// TIA Portal V20 export
// export: Created 2026-04-11T06:02:30.3000728Z, ExportSetting WithDefaults, DisplayName Totally Integrated Automation Portal, DisplayVersion V20, DisplayName TIA Portal Openness, DisplayVersion V20, DisplayName TIA Portal Version Control Interface, DisplayVersion V20, DisplayName STEP 7 Professional, DisplayVersion V20, DisplayName STEP 7 Safety, DisplayVersion V20, DisplayName WinCC Basic/Comfort/Advanced, DisplayVersion V20, DisplayName WinCC Unified, DisplayVersion V20
TYPE "udtHMI_AnalogValveControl"
// stored: IsFailsafeCompliant false
   STRUCT
      iMode : Int;   // Current mode
      iErrorCode { ExternalWritable := 'False'} : Int;   // Error code
      iStatus { ExternalWritable := 'False'} : Int;   // Color status for HMI
      rManualSP { S7_SetPoint := 'True'} : Real;   // Set point for manual mode
      rAutoSP { ExternalWritable := 'False'} : Real;   // Set point for automatic mode
      rEstopSP { S7_SetPoint := 'True'} : Real;   // Set point for an e-stop condition, if selected
      rActual { ExternalWritable := 'False'} : Real;   // Actual value
      bPB_ResetError : Bool;   // PB Reset errors
      bPBEN_ResetError { ExternalWritable := 'False'} : Bool;   // PB reset errors enable
      bError { ExternalWritable := 'False'} : Bool;   // Overall error
      bInterlock { ExternalWritable := 'False'} : Bool;   // Valve Interlocked
      iEstopFunction { S7_SetPoint := 'True'} : Int;   // Enum of E-Stop repsonse (Estop.xxx)
   END_STRUCT;
END_TYPE
